Fanuc KAREL source: pathswrapper.klc

PROGRAM class_name
%NOBUSYLAMP
%COMMENT = 'paths wrapper'
%NOLOCKGROUP

%include namespace.m

%include systemlib.klt
%include systemvars.klt
%include pose.const.klt
%include draw.klt
%include paths.klt
%include toolpath.structs.klt
%include pathswrapper.deps.klt

%define BASE_CLASSNAME class_name

VAR
  bbox : t_RECT
  contours : PATH nodedata = t_VEC_PATH
  lines : PATH nodedata = t_VEC_PATH

%from systemlib.klh %import VEC, VEC2D
%from pose.klh %import set_config
%include paths.klh

--define objects
  --polygon
draw_object_define(DRAW_OBJECT_NAME,CONFIG_FILENAME)

%defeval class_name BASE_CLASSNAME

%include pathswrapper.klh
%include pathswrapper.private.klh

--private

ROUTINE raster
  BEGIN
    --get raster lines
    -- (start_angle, dir, wall_lines, line_width, line_pitch)
    `DRAW_OBJECT_NAME`__set_params((rastprm.angle), (rastprm.dir), (rastprm.contours), &
                                   (rastprm.line_width), (rastprm.overlap) )
    `DRAW_OBJECT_NAME`__raster(PTH_LINETO)

    paths__clear_vecpath(lines) ; paths__clear_vecpath(contours) ;

    --get lines from object
    `DRAW_OBJECT_NAME`__lines_to_vec_path(lines) ;
    `DRAW_OBJECT_NAME`__contours_to_vec_path(contours) ;
    --get bounding box
    bbox = `DRAW_OBJECT_NAME`__get_bounding_box

  END raster

--public

ROUTINE delete
  BEGIN
    --clear wrapper members
    paths__clear_vecpath(contours)
    paths__clear_vecpath(lines)

    --clear draw object
    `DRAW_OBJECT_NAME`__delete
  END delete

ROUTINE get_lines
  VAR
    status : INTEGER
  BEGIN
    COPY_PATH(lines, 0, 0, out_lines, status)
  END get_lines

ROUTINE get_contours
  VAR
    status : INTEGER
  BEGIN
    COPY_PATH(contours, 0, 0, out_contour, status)
  END get_contours


ROUTINE drawPad
  BEGIN
    --draw pads
    `DRAW_OBJECT_NAME`__new
    `DRAW_OBJECT_NAME`__pads(padprm.width, padprm.length, padprm.separation, padprm.no_of_pads, VEC2D(0,0))

    --raster shape
    raster(rastprm)

  END drawPad

ROUTINE drawHex
  BEGIN
    --draw pads
    `DRAW_OBJECT_NAME`__new
    `DRAW_OBJECT_NAME`__hexagon((hexprm.radius), (hexprm.points), VEC2D(0, 0), (polyprm.polyRotation))

    --raster shape
    raster(rastprm)

  END drawHex

ROUTINE drawCustom
  VAR
    p : XYZWPR
  BEGIN

    --draw pads
    `DRAW_OBJECT_NAME`__new
    --apply polygon z-rotation to input frame
    p = poly_frame:POS(0,0,0,0,0,(polyprm.polyRotation),poly_frame.Config_data)
    `DRAW_OBJECT_NAME`__set_canvas(p)
    `DRAW_OBJECT_NAME`__import_shape('FR:\' + filename + '.csv')

    --raster shape
    raster(rastprm)

  END drawCustom

BEGIN
END class_name
